// TwinCAT 3 PLC project PLC
// Title: SPT Component Template
// Company: Beckhoff Automation LLC
// Author: F. Simmel
// ProjectVersion: 1.0.0
// ProgramVersion: 3.1.4024.0
// libraries:
//   SPT Base Types, * (Beckhoff Automation LLC)
//   SPT Event Logger, * (Beckhoff Automation LLC)
//   Tc2_Standard, * (Beckhoff Automation GmbH)
//   Tc2_System, * (Beckhoff Automation GmbH)
//   Tc3_EventLogger, * (Beckhoff Automation GmbH)
//   Tc3_Module, * (Beckhoff Automation GmbH)
//   Tc3_PackML_V2, * (Beckhoff Automation GmbH)
// project tree:
//   Machine/Components/MyComponent/DUTs/HMI/ ST_ComponentMyComponent_Command.TcDUT, ST_ComponentMyComponent_Config.TcDUT, ST_ComponentMyComponent_HMI.TcDUT, ST_ComponentMyComponent_Status.TcDUT
//   Machine/Components/MyComponent/ FB_Component_MyComponent.TcPOU
//   Machine/Components/MyComponent/Interfaces/ I_MyComponent.TcIO
//   Machine/ FB_Machine.TcPOU
//   / MAIN.TcPOU, PlcTask.TcTTO
// real-time tasks:
//   TASK PlcTask: cycle T#10ms, priority 20, ADS port 350

CONFIGURATION PLC
    RESOURCE PLC ON TwinCAT3
        TASK PlcTask(INTERVAL := T#10ms, PRIORITY := 20);
        PROGRAM MAIN WITH PlcTask : MAIN;
    END_RESOURCE
END_CONFIGURATION

// ---- Machine/Components/MyComponent/DUTs/HMI/ST_ComponentMyComponent_Command.TcDUT
TYPE ST_ComponentMyComponent_Command :
	STRUCT
		MyCommand1 : BOOL;
		MyCommand2 : BOOL;
	END_STRUCT
END_TYPE

// ---- Machine/Components/MyComponent/DUTs/HMI/ST_ComponentMyComponent_Config.TcDUT
TYPE ST_ComponentMyComponent_Config :
	STRUCT
	END_STRUCT
END_TYPE

// ---- Machine/Components/MyComponent/DUTs/HMI/ST_ComponentMyComponent_HMI.TcDUT
TYPE ST_ComponentMyComponent_HMI :
	STRUCT
		Config	: ST_ComponentMyComponent_Config;  // Settings e.g. Timeout, IP Address,...
		Command : ST_ComponentMyComponent_Command; // Command to be execute from HMI e.g. extend, retract,...
		Status	: ST_ComponentMyComponent_Status;  // Feedback from Component to HMI e.g. extended, retracted,...
	END_STRUCT
END_TYPE

// ---- Machine/Components/MyComponent/DUTs/HMI/ST_ComponentMyComponent_Status.TcDUT
TYPE ST_ComponentMyComponent_Status :
	STRUCT
		MyVarProperty1 : BOOL;
		MyVarProperty2 : BOOL;
	END_STRUCT
END_TYPE

// ---- Machine/Components/MyComponent/Interfaces/I_MyComponent.TcIO
INTERFACE I_MyComponent EXTENDS I_BaseFB

METHOD MyCommand1 : BOOL
VAR_INPUT
END_VAR
END_METHOD

METHOD MyCommand2 : BOOL
VAR_INPUT
END_VAR
END_METHOD

PROPERTY MyVarProperty1 : BOOL
GET
END_GET
SET
END_SET
END_PROPERTY

PROPERTY MyVarProperty2 : BOOL
GET
END_GET
SET
END_SET
END_PROPERTY

END_INTERFACE

// ---- MAIN.TcPOU
PROGRAM MAIN
VAR
	Machine		 : FB_Machine := (Name := 'Machine');
	InitComplete : BOOL;
END_VAR

IF NOT InitComplete THEN
	InitComplete := Initialize();
	RETURN;
END_IF

//Machine Cyclic Logic
Machine.CyclicLogic();

METHOD Initialize : BOOL
VAR_INPUT
END_VAR
Initialize := TRUE;
END_METHOD

END_PROGRAM

// ---- Machine/FB_Machine.TcPOU
FUNCTION_BLOCK FB_Machine EXTENDS FB_PackML_BaseModule
VAR
	(*List of Components*)
	MyComponent : FB_Component_MyComponent := (Name := 'My Component');

	(*Alarms for this module*)
	MachineAlarms : ARRAY[1..MACHINE_ALARM_COUNT] OF FB_TcAlarm;
END_VAR

VAR CONSTANT
	//Alarm count constant
	MACHINE_ALARM_COUNT : INT := 1; //Change this value based on how many alarms are in your machine
END_VAR

METHOD PROTECTED Aborting
VAR
	i				: UDINT;
	SubModulesReady : BOOL := TRUE;
END_VAR
CASE _CurrentMode OF
	E_PMLUnitMode.ePMLUnitMode_Production, E_PMLUnitMode.ePMLUnitMode_Maintenance, E_PMLUnitMode.ePMLUnitMode_Manual:
		CASE SequenceState OF
			0:
				SUPER^.Aborting();
		END_CASE
END_CASE
END_METHOD

METHOD PROTECTED Clearing
VAR
	i				: UDINT;
	SubModulesReady : BOOL := TRUE;
END_VAR
CASE _CurrentMode OF
	//=================================PRODUCTION MODE==================================
	E_PMLUnitMode.ePMLUnitMode_Production:
		SUPER^.Clearing();

	//=================================MAINTENANCE MODE==================================	
	E_PMLUnitMode.ePMLUnitMode_Maintenance:
		SUPER^.Clearing();

	//=================================MANUAL MODE==================================
	E_PMLUnitMode.ePMLUnitMode_Manual:
		SUPER^.Clearing();
END_CASE
END_METHOD

//! @summary This method monitors <b>components</b> within this PackML module and initiates fault responses as required
METHOD PROTECTED ComponentMonitor : BOOL
VAR
	AlarmResponses : ARRAY[0..4] OF E_AlarmResponse; //Temporary response array
	i			   : UDINT;
END_VAR

//! @description This method is called cyclically by <c>CyclicLogic()</c>
Super^.ComponentMonitor();
END_METHOD

METHOD PROTECTED CreateEvents
VAR_INPUT
END_VAR
// Add your event creation here
F_CreateAllEventsInClass(Alarms		:= MachineAlarms,
						 ClassSize	:= SIZEOF(TC_Events.Machine),
						 pInitEvent := ADR(TC_EVENTS.Machine.InitReferenceEvent),
						 Prefix		:= Name);

// Super call to base
SUPER^.CreateEvents();
END_METHOD

METHOD CyclicLogic
VAR_INPUT
END_VAR
IF NOT _InitComplete THEN
	_InitComplete := Initialize();
	RETURN;
END_IF

(* Inhibit Cylinder Movmements *)

(* Call Super *)
SUPER^.CyclicLogic();
CyclicLogic_Monitoring();
END_METHOD

METHOD PROTECTED CyclicLogic_Monitoring
VAR_INPUT
END_VAR
(*	
Monitor machine alarms here
*)

(*IF EstopInput1 AND NOT MachineAlarms[E_PLC1.EmergencyStop1].bRaised THEN
    RaiseAlarmWithStrings(MachineAlarms[E_PLC1.EmergencyStop1], '', '');
ELSIF NOT EstopInput1 AND MachineAlarms[E_PLC1.EmergencyStop1].bRaised THEN
    MachineAlarms[E_PLC1.EmergencyStop1].Clear(0, 0);
END_IF*)
END_METHOD

METHOD PROTECTED FINAL Execute
CASE _CurrentMode OF
	//=================================PRODUCTION MODE==================================
	E_PMLUnitMode.ePMLUnitMode_Production:
		CASE SequenceState OF
			0:
		END_CASE

	//=================================MAINTENANCE MODE==================================	
	E_PMLUnitMode.ePMLUnitMode_Maintenance:

	//=================================MANUAL MODE==================================
	E_PMLUnitMode.ePMLUnitMode_Manual:
END_CASE
END_METHOD

METHOD PROTECTED HMIPermissions
VAR_INPUT
END_VAR
CASE _CurrentMode OF
	//=================================PRODUCTION MODE==================================
	E_PMLUnitMode.ePMLUnitMode_Production:
		AllowHMIControl(ThisModuleOnly := TRUE);

	//=================================MAINTENANCE MODE==================================	
	E_PMLUnitMode.ePMLUnitMode_Maintenance:
		AllowHMIControl(ThisModuleOnly := FALSE);

	//=================================MANUAL MODE==================================
	E_PMLUnitMode.ePMLUnitMode_Manual:
		AllowHMIControl(ThisModuleOnly := FALSE);
END_CASE
END_METHOD

METHOD PROTECTED Initialize : BOOL
VAR
	i : UDINT; //Generic iteration value
END_VAR
Initialize := FALSE;
CASE DescendantSequenceState OF
	0:
		//RegisterComponent(Servo);
		_LogModeChanges			:= FALSE;
		_LogStateChanges		:= FALSE;
		DescendantSequenceState := DescendantSequenceState + 10;

	10:
		//Setup Custom modes here
		CustomModes(eMode						   := E_PMLUnitMode.ePMLUnitMode_Production,
					sName						   := 'Production',
					bDisableClearing			   := FALSE,
					bDisableStarting			   := FALSE,
					bDisableSuspended			   := TRUE,
					bDisableStopping			   := FALSE,
					bDisableAborting			   := FALSE,
					bDisableHolding				   := TRUE,
					bDisableHeld				   := TRUE,
					bDisableUnholding			   := TRUE,
					bDisableSuspending			   := TRUE,
					bDisableUnsuspending		   := TRUE,
					bDisableResetting			   := TRUE,
					bDisableIdle				   := TRUE,
					bDisableCompleting			   := TRUE,
					bDisableComplete			   := TRUE,
					bEnableUnitModeChangeStopped   := TRUE,
					bEnableUnitModeChangeIdle	   := TRUE,
					bEnableUnitModeChangeSuspended := FALSE,
					bEnableUnitModeChangeExecute   := FALSE,
					bEnableUnitModeChangeAborted   := TRUE,
					bEnableUnitModeChangeHeld	   := FALSE,
					bEnableUnitModeChangeComplete  := TRUE,
					bError						   =>,
					nErrorId					   =>);

		CustomModes(eMode						   := E_PMLUnitMode.ePMLUnitMode_Manual,
					sName						   := 'Manual',
					bDisableClearing			   := FALSE,
					bDisableStarting			   := FALSE,
					bDisableSuspended			   := TRUE,
					bDisableStopping			   := FALSE,
					bDisableAborting			   := FALSE,
					bDisableHolding				   := TRUE,
					bDisableHeld				   := TRUE,
					bDisableUnholding			   := TRUE,
					bDisableSuspending			   := TRUE,
					bDisableUnsuspending		   := TRUE,
					bDisableResetting			   := TRUE,
					bDisableIdle				   := TRUE,
					bDisableCompleting			   := TRUE,
					bDisableComplete			   := TRUE,
					bEnableUnitModeChangeStopped   := TRUE,
					bEnableUnitModeChangeIdle	   := TRUE,
					bEnableUnitModeChangeSuspended := TRUE,
					bEnableUnitModeChangeExecute   := TRUE,
					bEnableUnitModeChangeAborted   := TRUE,
					bEnableUnitModeChangeHeld	   := TRUE,
					bEnableUnitModeChangeComplete  := TRUE,
					bError						   =>,
					nErrorId					   =>);

		CustomModes(eMode						   := E_PMLUnitMode.ePMLUnitMode_Maintenance,
					sName						   := 'Maintenance',
					bDisableClearing			   := FALSE,
					bDisableStarting			   := FALSE,
					bDisableSuspended			   := TRUE,
					bDisableStopping			   := FALSE,
					bDisableAborting			   := FALSE,
					bDisableHolding				   := TRUE,
					bDisableHeld				   := TRUE,
					bDisableUnholding			   := TRUE,
					bDisableSuspending			   := TRUE,
					bDisableUnsuspending		   := TRUE,
					bDisableResetting			   := TRUE,
					bDisableIdle				   := TRUE,
					bDisableCompleting			   := TRUE,
					bDisableComplete			   := TRUE,
					bEnableUnitModeChangeStopped   := TRUE,
					bEnableUnitModeChangeIdle	   := TRUE,
					bEnableUnitModeChangeSuspended := TRUE,
					bEnableUnitModeChangeExecute   := TRUE,
					bEnableUnitModeChangeAborted   := TRUE,
					bEnableUnitModeChangeHeld	   := TRUE,
					bEnableUnitModeChangeComplete  := TRUE,
					bError						   =>,
					nErrorId					   =>);

		DescendantSequenceState := DescendantSequenceState + 10;

	20:
		//Copy Mode names
		FOR i := 1 TO 3 DO
			ModeNames[i] := F_UnitModeToString(UDINT_TO_DINT(i));
		END_FOR

		DescendantSequenceState := DescendantSequenceState + 10;

	30:
		// Initialize Recipes 
		DescendantSequenceState := DescendantSequenceState + 10;

	40:
		//Call the Super
		IF SUPER^.Initialize() THEN
			DescendantSequenceState := DescendantSequenceState + 10;
		END_IF

	50:
		Initialize := TRUE;
END_CASE
END_METHOD

METHOD PROTECTED Starting
VAR
	i				: UDINT;
	SubModulesReady : BOOL := TRUE;
END_VAR
CASE _CurrentMode OF
	E_PMLUnitMode.ePMLUnitMode_Production, E_PMLUnitMode.ePMLUnitMode_Maintenance, E_PMLUnitMode.ePMLUnitMode_Manual:
		CASE SequenceState OF
			0:
				SUPER^.Starting();
		END_CASE
END_CASE
END_METHOD

//! @summary This method contains code which will execute when this PackML module is in the <b>Stopping</b> state
METHOD PROTECTED Stopping
VAR
	i				: UDINT;
	SubModulesReady : BOOL := TRUE;
END_VAR

(*! <description><b></b><table> 
	<tr>
		<th> Previous State </th>
		<th> Transition In </th>
		<th> Transition Out </th>
		<th> Next State  </th> 
	</tr>
	<tr>
		<td> <b>ANY<i>except</i></b>Stopped<b>-or-</b>Clearing<b>-or-</b>Aborted<b>-or-</b>Aborting</td>
		<td> Stop Command </td> 
		<td> State Complete </td>
		<td> Stopped </td> 
	</tr>
</table>
This method is called as required by <c>StateControl()</c>
</description> 

*)
CASE _CurrentMode OF
	E_PMLUnitMode.ePMLUnitMode_Production, E_PMLUnitMode.ePMLUnitMode_Maintenance, E_PMLUnitMode.ePMLUnitMode_Manual:
		CASE SequenceState OF
			0:
				SUPER^.Stopping();
		END_CASE
END_CASE
END_METHOD

METHOD PROTECTED SubModuleMonitor : BOOL
VAR
	AlarmResponses : ARRAY[0..4] OF E_AlarmResponse; //Temporary response array	
END_VAR
// Check the sub Modules for Alarm Severity
SUPER^.SubModuleMonitor();

//Check the alarms at the machine level
_CurrentAlarmSeverity := F_GetMaxSeverityRaised(Alarms := MachineAlarms, CurrentSeverity := _CurrentAlarmSeverity);

//Check the severity of the machine level alarms
IF _CurrentState <> E_PMLState.ePMLState_Aborted AND _CurrentState <> E_PMLState.ePMLState_Aborting AND _CurrentState <> E_PMLState.ePMLState_Clearing AND _CurrentState <> E_PMLState.ePMLState_Stopped AND _CurrentState <> E_PMLState.ePMLState_Stopping THEN
	AlarmResponses := _ParentFaultResponseDefinitions;
	CASE AlarmResponses[CurrentAlarmSeverity] OF
		E_AlarmResponse.Abort_ImmediateError:
			AbortImmediateError(Name, TRUE);

		E_AlarmResponse.Abort_Immediate:
			AbortImmediate();

		E_AlarmResponse.Stop_Immediate:
			StopImmediate();

		E_AlarmResponse.Stop_Controlled:
			StopControlled();

		E_AlarmResponse.Hold_Immediate:
			HoldImmediate();

		E_AlarmResponse.Suspend_Immediate:
			SuspendImmediate();

		E_AlarmResponse.Suspend_Controlled:
			SuspendControlled();

		E_AlarmResponse.NoResponse:
			;
	END_CASE
ELSIF _CurrentState = E_PMLState.ePMLState_Stopped OR _CurrentState = E_PMLState.ePMLState_Stopping THEN
	AlarmResponses := _ParentFaultResponseDefinitions;
	CASE AlarmResponses[CurrentAlarmSeverity] OF
		E_AlarmResponse.Abort_ImmediateError:
			AbortImmediateError(Name, TRUE);

		E_AlarmResponse.Abort_Immediate:
			AbortImmediate();

		E_AlarmResponse.NoResponse:
			;
	END_CASE
END_IF
END_METHOD

END_FUNCTION_BLOCK

// ---- Machine/Components/MyComponent/FB_Component_MyComponent.TcPOU
FUNCTION_BLOCK FB_Component_MyComponent EXTENDS FB_ComponentBase IMPLEMENTS I_MyComponent
VAR
	{error 'Programming instruction - Remove example variables'}

	// Inputs
	MyInput AT %I* : BOOL;

	// Outputs
	MyOutput AT %Q* : BOOL;

	// HMI
	MyComponent_HMI			: ST_ComponentMyComponent_HMI;
	HMICommandDescendant_RT : R_TRIG;

	// Alarms
	MyComponentAlarms : ARRAY[1..MY_COMPONENT_ALARMS_COUNT] OF FB_TcAlarm;

	// Internal variables
	_MyVarProperty1 : BOOL;
	_MyVarProperty2 : BOOL;
	MyVarInternal1	: BOOL;
	MyVarInternal2	: BOOL;

	//MyCommandFb		: MyCommandFB;// Command FB to execute something e.g. MC_MoveAbsolute
END_VAR

VAR CONSTANT
	MY_COMPONENT_ALARMS_COUNT : UDINT := 2;
END_VAR

// NO CODE HERE!!!

//! @summary Initializes event function blocks using this components's name
{attribute 'call_after_online_change_slot' := '<slot>'}
METHOD PROTECTED CreateEvents

//! @description This method is called by <c>Initialize()</c> as required
SUPER^.CreateEvents();
F_CreateAllEventsInClass(Alarms		:= MyComponentAlarms,
						 ClassSize	:= SIZEOF(TC_EVENTS.MyComponentAlarms),
						 pInitEvent := ADR(TC_EVENTS.MyComponentAlarms.InitReferenceEvent),
						 Prefix		:= _Name);
END_METHOD

//! @summary This method serves as the entry point for all underlying FB logic
METHOD PUBLIC CyclicLogic

//! @description This method should be called cyclically by descendant function blocks by invoking <c>SUPER^.CyclicLogic()</c>.  Alternatively, the contents of this method could be reimplemented entirely in which case a call to this method would not be necessary.
// Initialize Component
IF NOT _InitComplete THEN
	_InitComplete := Initialize();
	RETURN;
END_IF

{error 'Programming instruction - Write your custom component cyclic cogic here'}

(*
	MyCommandFb();
	IF MyCommandFB.Error THEN
		_Error	 := TRUE;
		_ErrorID := MyCommandFb.ErrorId;
	END_IF
	
	MyCommandFB.Execute := FALSE;
*)

// Component Error
{error 'Programming instruction - Create component has error'}
_Error	 := TRUE;
_ErrorID := 9999;

// Component Busy
{error 'Programming instruction - Create component is busy'}
IF TRUE THEN
	_Busy := TRUE;
ELSE
	_Busy := FALSE;
END_IF

// Call Super
SUPER^.CyclicLogic();

// Set Current Alarm Severity
_CurrentAlarmSeverity := F_GetMaxSeverityRaised(Alarms := MyComponentAlarms, CurrentSeverity := _CurrentAlarmSeverity);
END_METHOD

//! @summary Provides interlocks for HMI control and updates HMI status information for this component
METHOD PROTECTED HMICommunication

//! @description This method is called cyclically by <c>CyclicLogic()</c>
SUPER^.HMICommunication();
{error 'Programming instruction - Add HMI communication'}

//Process HMI requests
HMICommandDescendant_RT(CLK := (ComponentBase_HMI.Status.HMIControlAvailable AND NOT HMICommandActive_Base) AND (MyComponent_HMI.Command.MyCommand1 XOR MyComponent_HMI.Command.MyCommand2));

//Base components should observe this to interlock HMI commands
HMICommandActive_Descendant := ComponentBase_HMI.Status.HMIControlAvailable AND (MyComponent_HMI.Command.MyCommand1 OR MyComponent_HMI.Command.MyCommand2);
IF HMICommandDescendant_RT.Q THEN
	IF MyComponent_HMI.Command.MyCommand1 THEN
		MyCommand1();
	END_IF

	IF MyComponent_HMI.Command.MyCommand2 THEN
		MyCommand2();
	END_IF
END_IF

//Update HMI status info
MyComponent_HMI.Status.MyVarProperty1 := _MyVarProperty1;
MyComponent_HMI.Status.MyVarProperty2 := _MyVarProperty2;
END_METHOD

//! @summary Basic component initialization logic
METHOD PROTECTED Initialize : BOOL;

//! @description This method is called by <c>CyclicLogic()</c> as required
{error 'Programming instruction - Add code to initialize your Component'}

//

//

// Call Super after init of your Component is completed sucessfully

// Call Super
Initialize := Super^.Initialize();
END_METHOD

//! Provides basic error detection and event handling for this component
METHOD PROTECTED Monitoring

(*! @descriptionThis method is called cyclically by <c>CyclicLogic()</c>*)
SUPER^.Monitoring();
{error 'Programming instruction - Raise custom alarms here'}
IF TRUE AND NOT MyComponentAlarms[E_MyComponentAlarms.MyExampleError].bRaised THEN
	RaiseAlarmWithStrings(MyComponentAlarms[E_MyComponentAlarms.MyExampleError], '', '');
END_IF
END_METHOD

METHOD MyCommand1 : BOOL
// Component already busy -> return and not accept command
IF _Busy THEN
	// Trace Message Command was not accepted
	TRACE('MyCommand1 rejected, component busy!');
	RETURN;
END_IF

{error 'Programming instruction - Execute command here'}

// Execute MyCommand1.....

(*
	MyCommandFb.Execute := TRUE;
*)
{error 'Programming instruction - Return command accepted in same cycle'}
MyCommand1 := TRUE;
END_METHOD

METHOD MyCommand2 : BOOL
END_METHOD

PROPERTY MyVarProperty1 : BOOL
GET
MyVarProperty1 := _MyVarProperty1;
END_GET
SET
_MyVarProperty1 := MyVarProperty1;
END_SET
END_PROPERTY

PROPERTY MyVarProperty2 : BOOL
GET
MyVarProperty2 := _MyVarProperty2;
END_GET
SET
_MyVarProperty2 := MyVarProperty2;
END_SET
END_PROPERTY

//! @summary Clears error flags and error IDs for this component
METHOD PUBLIC Reset : BOOL
{error 'Programming instruction - Reset component here'}

//

//

//

// Clear Component Alarms
F_ClearAllEventsInClass(MyComponentAlarms);

// Call Super
Reset := Super^.Reset();
END_METHOD

END_FUNCTION_BLOCK
